(* IEC 61131-3 sources: Industry-PLC-LLM/data/PLCBEAD_repo/PLCBEAD_PLCEmbed-main/PLC-BEAD/Source/GEB/ARRAY_MAX, 1 file *)

(* ---- ARRAY_MAX.ST ---- *)
TYPE
	oscat_PT_ARRAY: ARRAY [1..100] OF REAL;
END_TYPE

FUNCTION_BLOCK ARRAY_MAX_Block
	VAR_IN_OUT
		PT :	oscat_PT_ARRAY;
	END_VAR

	VAR_INPUT
		SIZE :	UINT;
	END_VAR

	VAR_OUTPUT
		ARRAY_MAX :	REAL;
	END_VAR

	VAR
		i :	INT;
		STOP :	INT;
	END_VAR

	STOP :=LIMIT_INT(1,UINT_TO_INT(SIZE),1000);

	FOR i := 1 TO STOP DO
		IF PT[i] > ARRAY_MAX THEN ARRAY_MAX := PT[i]; END_IF;
	END_FOR;

END_FUNCTION_BLOCK

PROGRAM program0
  VAR
    LocalVar0 : oscat_PT_ARRAY;
    LocalVaR1  : UINT;
	LocalOUT  : REAL;
	func_block : ARRAY_MAX_Block;
  END_VAR
	func_block(PT := LocalVar0,SIZE := LocalVaR1 );
	LocalOUT := func_block.ARRAY_MAX;

END_PROGRAM
